FUNCTION_BLOCK FB_TestChain2 EXTENDS FB_Chain
VAR_INPUT
END_VAR
VAR_OUTPUT
END_VAR
VAR
END_VAR

super^(io_fbChainController := io_fbChainController);

METHOD init : BOOL
VAR_INPUT
END_VAR
CASE initStep OF
0:

10:
	io_fbChainController.releaseForChain(sChainToRelease := 'fbChain1',THIS^);
	initStep := 20;
20:

30:

END_CASE
END_METHOD

END_FUNCTION_BLOCK

(* stored: Version 1.1.0.1, ProductVersion 3.1.4024.0
   POU FB_TestChain2: Id {1f2848b6-6170-45e2-b2f6-0f3a28090b40}, SpecialFunc None
   Method init: Id {438c0a1d-f1f3-47de-9174-4ef5d89284e7} *)
